FUNCTION_BLOCK EL3413
VAR
	_io : EL3413_Data;
	{attribute addProperty Name "WcState"}
	_wcState : WcStateInputToggle;
	{attribute addProperty Name "Info data"}
	_infoData : InfoDataAds;
END_VAR

PROPERTY IO : REFERENCE TO EL3413_Data
GET
IO REF= _io;
END_GET
END_PROPERTY

PROPERTY WcState : REFERENCE TO WcStateInputToggle
GET
WcState REF= _wcState;
END_GET
END_PROPERTY

END_FUNCTION_BLOCK

(* stored: Version 1.1.0.1, ProductVersion 3.1.4024.9
   POU EL3413: Id {69b112a8-50aa-0790-1859-0574338231fc}, SpecialFunc None
   Property IO: Id {90fc9e8c-a50b-0ad6-39e1-a424beac33c6}
   Get Get: Id {3216bb97-8019-07df-2504-82f9193f3c1b}
   Property WcState: Id {43c0707c-e70d-0c18-2d19-d033ef908a72}
   Get Get: Id {01219d49-c5a3-03a6-1444-bc715b42b660} *)
